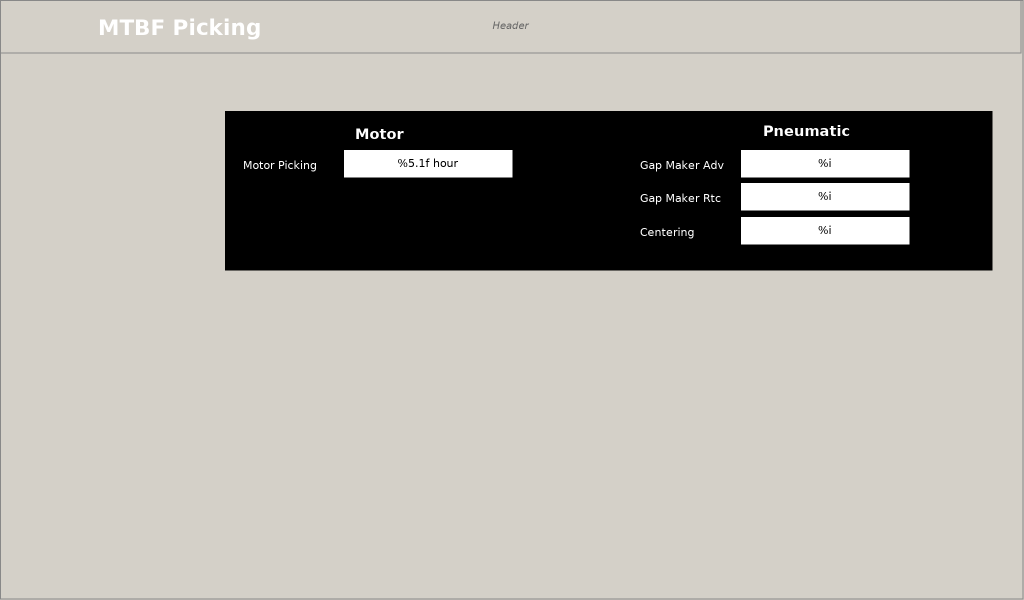
VISUALIZATION MTBF_Picking  // 1024x600
    Frame (0,-2 1021x55)
        shows Header()
    Label (95,15 250x25), "MTBF Picking"
    RoundedRectangle (225,111 767x159)
    Label (243,114 273x40), "Motor"
    Label (240,148 103x35), "Motor Picking"
    RoundedRectangle (343,149 170x29), "%5.1f hour", text variable: Status_GVL.stMotor_Picking.RunningHours
    Label (637,148 104x35), "Gap Maker Adv"
    RoundedRectangle (740,149 170x29), "%i", text variable: Status_GVL.stPneu_GapMaker.CyclePneuAdv
    Label (670,111 273x40), "Pneumatic"
    Label (637,181 104x35), "Gap Maker Rtc"
    RoundedRectangle (740,182 170x29), "%i", text variable: Status_GVL.stPneu_GapMaker.CyclePneuRtc
    Label (637,215 104x35), "Centering"
    RoundedRectangle (740,216 170x29), "%i", text variable: Status_GVL.stPneu_Centering.CyclePneu
END_VISUALIZATION

(* stored: Version 1.1.0.1, ProductVersion 3.1.4024.12
   Visu MTBF_Picking: Id {c70a7542-8d2e-47a4-80d9-e218a662d99e} *)
